// Mitsubishi GX Works2 project: D1 메모리   PLC: Q02/Q02H

PROGRAM MAIN
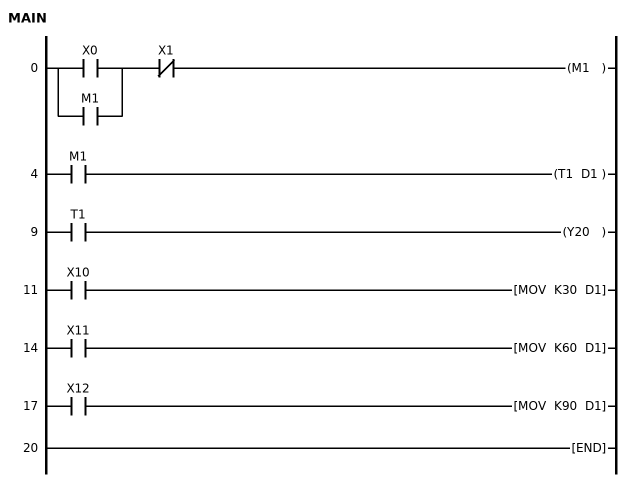
0     LD      X0
      OR      M1
      ANI     X1
      OUT     M1
4     LD      M1
      OUT     T1 D1
9     LD      T1
      OUT     Y20
11    LD      X10
      MOV     K30 D1
14    LD      X11
      MOV     K60 D1
17    LD      X12
      MOV     K90 D1
20    END
END_PROGRAM
